TYPE ST_Chamber1PreparePositionParam :
STRUCT
	LiftReady : ST_Chamber1LiftPinAxisMoveAbsParam;
	SpinAlign : ST_Chamber1SpinAxisMoveAbsParam;
	LiftWork : ST_Chamber1LiftPinAxisMoveAbsParam;
END_STRUCT
END_TYPE

(* stored: Version 1.1.0.1, ProductVersion 3.1.4026.18
   DUT ST_Chamber1PreparePositionParam: Id {c2f5cf23-dcac-4e62-b667-372e33e8180b} *)
